// TIA Portal V17 export
// export: Created 2025-03-05T08:01:25.5940182Z, ExportSetting WithDefaults, DisplayName Totally Integrated Automation Portal, DisplayVersion V17 Update 8, DisplayName TIA Portal Openness, DisplayVersion V17 Update 8, DisplayName TIA Portal Version Control Interface, DisplayVersion V17, DisplayName SINAMICS Startdrive Advanced, DisplayVersion V17 SP2, DisplayName SINAMICS Startdrive G110M, G120, G120C, G120D, G120P, G115D, DisplayVersion V17 SP2, DisplayName SINAMICS Startdrive G130, G150, S120, S150, SINAMICS MV, S210, DisplayVersion V17 SP2, DisplayName STEP 7 Professional, DisplayVersion V17 Update 8, DisplayName SINUMERIK ONE STEP 7 Toolbox, DisplayVersion V17 Update 12, DisplayName SINUMERIK 840D sl STEP 7 Toolbox, DisplayVersion V17 Update 12, DisplayName STEP 7 Safety, DisplayVersion V17 Update 6, DisplayName WinCC Advanced, DisplayVersion V17 Update 8
DATA_BLOCK "DB20301_LASER_GUIDE_UNIT_02"   // DB20301
{ DB_Accessible_From_OPC_UA := 'FALSE' }
VERSION : 0.1
// stored: AutoNumber false, DBAccessibleFromOPCUA false, DBAccessibleFromWebserver true, InstanceOfName FB20300_LASER_GUIDE, InstanceOfType FB
"FB20300_LASER_GUIDE"
   // VAR_INPUT
   //    iCONTROL_ON_DELAYED : Bool;
   //    iLASER_ACTIVE_LASER_ON : Bool;
   //    iSTART_MANUAL_REQUEST : Bool;
   //    iSTART_AUTO_REQUEST : Bool;
   //    iGUIDE_LASER_IS_ON : Bool;
   //    iSTOP_MANUAL_REQUEST : Bool;
   //    iSTOP_AUTO_REQUEST : Bool;
   //    iHOME_SEQUENCE_RUNNING : Bool;
   //    iCONTROL_OFF : Bool;
   //    TEMP : Timer;
   // END_VAR
   // VAR_OUTPUT
   //    oLASER_NOT_READY_ALARM : Bool;
   //    oSEOC_ALARMS : Bool;
   //    oSwitchoncondition_on : Bool;
   //    oSwitchoncondition_off : Bool;
   //    oMotion_Active_Right : Bool;
   //    oMotion_Active_Left : Bool;
   //    oLimit_right : Bool;
   //    oLimit_left : Bool;
   //    oGUIDE_LASER_ON : Bool;
   // END_VAR
   // VAR RETAIN
   //    DATA : "LASER GUIDE";
   // END_VAR
BEGIN
END_DATA_BLOCK
